// TIA Portal V18 export
TYPE "LGasp_typeRigaProdfromPLC"
// stored: IsFailsafeCompliant false
   STRUCT
      pzfatti : DInt;   // Pezzi completati (in punzonatura)
      pzfattinopasso : DInt;   // pezzi fatti non multipli del passo dello stampo / Pezzi fatti non a passo del feeder (in punzonatura)
      pzinseritinelriordinoquote : DInt;   // Pezzi presi in carico dal riordino quote
   END_STRUCT;
END_TYPE
